// TIA Portal V20 export
DATA_BLOCK "instGetIdentRf"   // DB165
// stored: InstanceOfName GetIdentRf, InstanceOfType FB
"GetIdentRf"
   // VAR_OUTPUT
   //    selectedRFID : USInt;
   //    selectedAntena : USInt;
   //    error : Word;
   // END_VAR
   // VAR_IN_OUT
   //    identRfAllUnits : Array[*] of "typeIdentRf";
   //    IdentRfInterfaceHmi : "typeIdentRfHmi";
   // END_VAR
   // VAR
   //    statSelectedRfReader : USInt;
   //    statSelectedAntena : USInt;
   // END_VAR
BEGIN
END_DATA_BLOCK
